(*
SPDX-FileCopyrightText: © 2026 Oleksandr Tiutyk <trofimich@gmail.com>
SPDX-License-Identifier: MIT
License: https://opensource.org/license/mit
*)

INTERFACE IStringOwerflowException EXTENDS IGeneralException

METHOD Throw
VAR_INPUT
	sourceNamespaceName : STRING;
	sourceClassName : STRING;
	sourcePOUName : STRING;
	sourcePosition : STRING;
	stringName : STRING;
	actualLength : UDINT;
	maxLength : UDINT;
END_VAR
END_METHOD

END_INTERFACE

(* stored: Version 1.1.0.1
   Itf IStringOwerflowException: Id {6a53b6ed-b7c4-44c9-9540-6a98d64ca74a}
   Method Throw: Id {370c5aa8-6645-4931-8e8b-bbe194df5099} *)
